FUNCTION_BLOCK AsyncResponseMiddleware EXTENDS MiddlewareBase
VAR
	asyncResponseManager : I_AsyncResponseManager;
END_VAR

METHOD FB_init : BOOL
VAR_INPUT
	bInitRetains : BOOL; // if TRUE, the retain variables are initialized (warm start / cold start)
	bInCopyCode : BOOL;  // if TRUE, the instance afterwards gets moved into the copy code (online change)
	AsyncResponseManager : I_AsyncResponseManager;
END_VAR
This^.asyncResponseManager := AsyncResponseManager;
END_METHOD

METHOD PUBLIC Handle
VAR_INPUT
	Request : I_Request;
	Response : I_ServerResponse;
END_VAR
IF asyncResponseManager.TryHandleIncomingRequest(Request, Response) THEN
	RETURN;
END_IF

Next(Request, Response);
END_METHOD

END_FUNCTION_BLOCK

(* stored: Version 1.1.0.1, ProductVersion 3.1.4026.13
   POU AsyncResponseMiddleware: Id {16b90780-5f51-4351-a7b2-cef2b626d16b}, SpecialFunc None
   Folder Constructor: Id {cc9bbf46-e628-41d7-8197-dfe9f8e61d29}
   Method FB_init: Id {266b3b21-04d6-41ff-a9e3-912a341b099e}
   Method Handle: Id {27f7a27b-bd24-444d-bbd1-48588c773a98} *)
